FUNCTION_BLOCK ColourSelect_V3 (* Template for a simple Basic Function Block Type *)
  (* Standard: 61499-2 *)
  (* Version 1.0, 2019-06-07, Promok *)
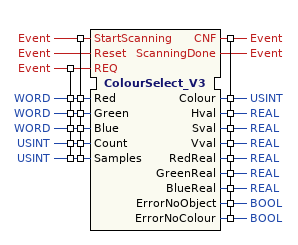
  EVENT_INPUT
    StartScanning WITH Red, Green, Blue, Samples, Count;
    Reset;
    REQ WITH Red, Green, Blue, Count, Samples; (* Normal Execution Request *)
  END_EVENT
  EVENT_OUTPUT
    CNF WITH ErrorNoObject, Colour, Vval, Sval, Hval, BlueReal, RedReal, GreenReal, ErrorNoColour;
    ScanningDone;
  END_EVENT
  VAR_INPUT
    Red : WORD; (* Input event qualifier *)
    Green : WORD;
    Blue : WORD;
    Count : USINT;
    Samples : USINT;
  END_VAR
  VAR_OUTPUT
    Colour : USINT;
    Hval : REAL;
    Sval : REAL;
    Vval : REAL;
    RedReal : REAL;
    GreenReal : REAL;
    BlueReal : REAL;
    ErrorNoObject : BOOL;
    ErrorNoColour : BOOL;
  END_VAR
  VAR
    Counter1 : USINT; (* Internal Variable *)
    Counter2 : USINT; (* Internal Variable *)
    Counter3 : USINT; (* Internal Variable *)
    Counter4 : USINT; (* Internal Variable *)
    Counter5 : USINT; (* Internal Variable *)
    ColourRecognized : BOOL; (* Internal Variable *)
    ObjectRecognized : BOOL; (* Internal Variable *)
    SamplesCounter : USINT; (* Internal Variable *)
    ScanDone : BOOL; (* Internal Variable *)
    Error : BOOL; (* Internal Variable *)
  END_VAR
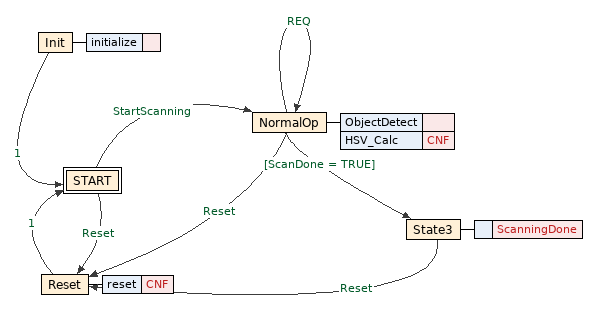
  EC_STATES
    START; (* Initial State *)
    NormalOp : ObjectDetect, HSV_Calc -> CNF; (* Normal execution *)
    Init : initialize;
    Reset : reset -> CNF;
    State3 : -> ScanningDone;
  END_STATES
  EC_TRANSITIONS
    START TO NormalOp := StartScanning;
    Init TO START := 1;
    START TO Reset := Reset;
    Reset TO START := 1;
    NormalOp TO State3 := [ScanDone = TRUE];
    NormalOp TO NormalOp := REQ;
    State3 TO Reset := Reset;
    NormalOp TO Reset := Reset;
  END_TRANSITIONS
  ALGORITHM ObjectDetect IN ST: (* new algorithm *)
IF Red>= 30 AND  Green >=10 AND Blue >=10 THEN
	ErrorNoObject := FALSE;
ELSE
	ErrorNoObject := TRUE;

END_IF;
  END_ALGORITHM
  ALGORITHM initialize IN ST: (* new algorithm *)
ErrorNoColour := FALSE;
ErrorNoObject := FALSE;
  END_ALGORITHM
  ALGORITHM reset IN ST: (* new algorithm *)
ErrorNoColour := FALSE;
ErrorNoObject := FALSE;
Error := FALSE;
SamplesCounter := 0;

ScanDone := FALSE;

ColourRecognized := FALSE;

Counter1 := 0;
Counter2 := 0;
Counter3 := 0;
Counter4 := 0;
Counter5 := 0;
  END_ALGORITHM
  ALGORITHM HSV_Calc IN ST: (* new algorithm *)
VAR
Min: REAL;
Max: REAL;
Delta : REAL;

END_VAR;

RedReal := Red;
GreenReal := Green;
BlueReal := Blue;

IF Red <= Green  AND Red <= Blue THEN
	Min := Red;
ELSIF Green <= Red  AND Green <= Blue THEN
	Min := Green;
ELSE
	Min := Blue;
END_IF;

IF Red >= Green  AND Red >= Blue THEN
	Max := Red;
ELSIF Green >= Red  AND Green >= Blue THEN
	Max := Green;
ELSE
	Max := Blue;
END_IF;

Delta := Max - Min;

IF Max = 0 THEN
	Sval := 0;
ELSE
	Sval := Delta / Max;
END_IF;

IF Sval = 0 THEN
	Hval := 0;
ELSE
	IF Red = Max THEN
		Hval := (Green-Blue)/Delta;
	ELSIF Green = Max THEN
		Hval := (Blue - Red)/Delta;
	ELSIF Blue = Max THEN
		Hval := (Red - Green)/Delta;
	END_IF;

	Hval := Hval *60;

	IF Hval < 0 THEN
		Hval := Hval +360;
	END_IF;
END_IF;

Vval := Max;
Sval := Sval * 100;


IF Hval >=  350 AND Hval <= 360 AND Sval >= 80 AND Sval <=  90 THEN
	Counter1 := Counter1 +1;
	Counter5 := 0;
	Counter2 := 0;
	Counter3 := 0;
	Counter4 := 0;

ELSIF Hval >=  5 AND Hval <= 15 AND Sval >= 75 AND Sval <=  90 THEN
 	Counter2 := Counter2 +1;
 	Counter1 := 0;
	Counter5 := 0;
	Counter3 := 0;
	Counter4 := 0;

ELSIF Hval >=  22 AND Hval <= 35 AND Sval >= 80 AND Sval <=  90 THEN
 	Counter3 := Counter3 +1;
 	Counter1 := 0;
	Counter2 := 0;
	Counter5 := 0;
	Counter4 := 0;

ELSIF Hval >=  325 AND Hval <= 345 AND Sval >= 80 AND Sval <=  90 THEN
Counter4 := Counter4 +1;
	Counter1 := 0;
	Counter2 := 0;
	Counter3 := 0;
	Counter5 := 0;

ELSIF Hval >=  0 AND Hval <= 45 AND Sval >= 20 AND Sval <=  40 THEN
	Counter5 := Counter5 +1;
	Counter1 := 0;
	Counter2 := 0;
	Counter3 := 0;
	Counter4 := 0;
(*ELSE
 	Counter1 := 0;
	Counter2 := 0;
	Counter3 := 0;
	Counter4 := 0;
	Counter5 := 0;*)
END_IF;

IF Error THEN
	Counter1 := 0;
	Counter2 := 0;
	Counter3 := 0;
	Counter4 := 0;
	Counter5 := 0;
END_IF;


IF  ColourRecognized = FALSE AND Error = FALSE THEN

IF Counter1 >= Count THEN
	//ColourAlreadyDetected := TRUE;
	ColourRecognized := TRUE;
    Counter1 := 0;
	Counter2 := 0;
	Counter3 := 0;
	Counter4 := 0;
	Counter5 := 0;
	Colour := 1;

ELSIF Counter2 >= Count THEN
	//ColourAlreadyDetected := TRUE;
	ColourRecognized := TRUE;
    Counter1 := 0;
	Counter2 := 0;
	Counter3 := 0;
	Counter4 := 0;
	Counter5 := 0;
	Colour := 2;

ELSIF Counter3 >= Count THEN
	//ColourAlreadyDetected := TRUE;
	ColourRecognized := TRUE;
    Counter1 := 0;
	Counter2 := 0;
	Counter3 := 0;
	Counter4 := 0;
	Counter5 := 0;
	Colour := 3;

ELSIF Counter4 >= Count THEN
	//ColourAlreadyDetected := TRUE;
	ColourRecognized := TRUE;
    Counter1 := 0;
	Counter2 := 0;
	Counter3 := 0;
	Counter4 := 0;
	Counter5 := 0;
	Colour := 4;

ELSIF Counter5 >= Count THEN
	//ColourAlreadyDetected := TRUE;
	ColourRecognized := TRUE;
    Counter1 := 0;
	Counter2 := 0;
	Counter3 := 0;
	Counter4 := 0;
	Counter5 := 0;
	Colour := 5;

ELSE
 	Colour := 0;
 	ColourRecognized := FALSE;

END_IF;
END_IF;

IF ColourRecognized = FALSE AND SamplesCounter >= Samples THEN
	ErrorNoColour := TRUE;
	ScanDone := TRUE;

	ELSIF ColourRecognized = TRUE THEN
	ErrorNoColour := FALSE;
	ScanDone := TRUE;

END_IF;

IF ErrorNoColour OR ErrorNoObject THEN
	Error := TRUE;
END_IF;

SamplesCounter := SamplesCounter + 1;
  END_ALGORITHM
END_FUNCTION_BLOCK
